FUNCTION_BLOCK ABSTRACT ShutterBase EXTENDS TExecution IMPLEMENTS IDevice
VAR_INPUT
END_VAR
VAR_OUTPUT
END_VAR
VAR
	{attribute 'OPC.UA.DA' := '0'}
	_name : STRING;
	{attribute 'OPC.UA.DA' := '0'}
	_deviceID : STRING;				
	{attribute 'OPC.UA.DA' := '0'}	
	_family : DeviceFamily;	
	{attribute 'OPC.UA.DA' := '0'}
	_logger : Logger;
	{attribute 'OPC.UA.DA' := '0'}
	_message : StringBuilder;
	{attribute 'OPC.UA.DA' := '0'}
	_shutterConfig : DeviceConfiguration;	
END_VAR

PROPERTY DeviceID : STRING
GET
DeviceID := _deviceID;
END_GET
SET
_deviceID := DeviceID;
END_SET
END_PROPERTY

PROPERTY Family : DeviceFamily
GET
Family := _family;
END_GET
SET
_family := Family;
END_SET
END_PROPERTY

METHOD PROTECTED ABSTRACT ManualClose
VAR_INPUT
	Execute : BOOL;
END_VAR
END_METHOD

METHOD PROTECTED ABSTRACT ManualOpen
VAR_INPUT
	Execute : BOOL;
END_VAR
END_METHOD

PROPERTY Name : STRING
GET
Name := _name;
END_GET
SET
_name := Name;
END_SET
END_PROPERTY

END_FUNCTION_BLOCK

(* stored: Version 1.1.0.1, ProductVersion 3.1.4024.4
   POU ShutterBase: Id {b50ae82a-0ab6-41ce-bbec-09f22dfef17d}, SpecialFunc None
   Property DeviceID: Id {3320d7d8-2470-4d78-b002-0e1f2e07810b}
   Get Get: Id {8a570f02-6bb5-4991-9a81-fc20cd1a0eae}
   Set Set: Id {95d2c08e-9925-44b4-8558-081a568345cf}
   Property Family: Id {9804369d-8071-4e2c-82c3-605c621f84d1}
   Get Get: Id {6c6e7e55-5389-4738-83b9-863a59212a07}
   Set Set: Id {b39c2a7e-d313-4850-a0b3-ed046ab8a488}
   Method ManualClose: Id {f98d88b4-f05d-4ac7-b235-4ef3eb5a7182}
   Method ManualOpen: Id {d22989d3-ac27-42f8-80f9-383388aa72cc}
   Property Name: Id {94ddb3ec-0c25-46c1-923c-2690d50afccb}
   Get Get: Id {3bd12e72-19e8-490a-bdb9-dc0a4c2d5572}
   Set Set: Id {69061ac4-c8f4-4121-80da-cfc6fff43b40} *)
